FUNCTION_BLOCK ReactorLogic (* CAT Function Block Type *)
  (* Standard: 61499-2 *)
  (* Version 0.0, 6/7/2026, Schneider Electric, template *)
  PACKAGE SE.Nereda;
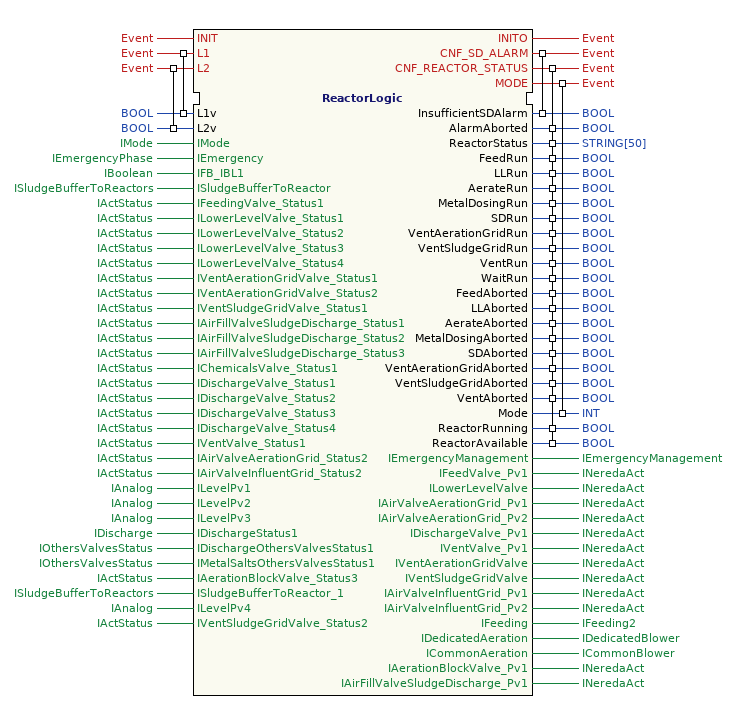
  EVENT_INPUT
    INIT;
    L1 WITH L1v;
    L2 WITH L2v;
  END_EVENT
  EVENT_OUTPUT
    INITO;
    CNF_SD_ALARM WITH InsufficientSDAlarm;
    CNF_REACTOR_STATUS WITH AlarmAborted, ReactorStatus, FeedRun, LLRun, AerateRun, MetalDosingRun, SDRun, VentAerationGridRun, VentSludgeGridRun, VentRun, WaitRun, FeedAborted, LLAborted, AerateAborted, MetalDosingAborted, SDAborted, VentAerationGridAborted, VentSludgeGridAborted, VentAborted, ReactorRunning, ReactorAvailable; (* Execution Confirmation *)
    MODE WITH Mode; (* Response from Socket *)
  END_EVENT
  VAR_INPUT
    L1v : BOOL;
    L2v : BOOL;
  END_VAR
  VAR_OUTPUT
    InsufficientSDAlarm : BOOL;
    AlarmAborted : BOOL; (* Result: IN1 OR IN2 OR ... *)
    ReactorStatus : STRING[50]; (* Output event qualifier *)
    FeedRun : BOOL;
    LLRun : BOOL;
    AerateRun : BOOL;
    MetalDosingRun : BOOL;
    SDRun : BOOL;
    VentAerationGridRun : BOOL;
    VentSludgeGridRun : BOOL;
    VentRun : BOOL;
    WaitRun : BOOL;
    FeedAborted : BOOL;
    LLAborted : BOOL;
    AerateAborted : BOOL;
    MetalDosingAborted : BOOL;
    SDAborted : BOOL;
    VentAerationGridAborted : BOOL;
    VentSludgeGridAborted : BOOL;
    VentAborted : BOOL;
    Mode : INT; (* Response Data from Socket *)
    ReactorRunning : BOOL; (* Result: IN1 OR IN2 OR ... *)
    ReactorAvailable : BOOL; (* Result: IN1 AND IN2 AND ... *)
  END_VAR
  SOCKETS
    IMode : IMode;
    IEmergency : IEmergencyPhase;
    IFB_IBL1 : IBoolean;
    ISludgeBufferToReactor : ISludgeBufferToReactors;
  END_SOCKETS
  SOCKETS
    IFeedingValve_Status1 : IActStatus; (* Phase Feed Status *)
    ILowerLevelValve_Status1 : IActStatus;
    ILowerLevelValve_Status2 : IActStatus;
    ILowerLevelValve_Status3 : IActStatus;
    ILowerLevelValve_Status4 : IActStatus;
    IVentAerationGridValve_Status1 : IActStatus;
    IVentAerationGridValve_Status2 : IActStatus; (* Phase Aerate Status *)
    IVentSludgeGridValve_Status1 : IActStatus;
    IAirFillValveSludgeDischarge_Status1 : IActStatus;
    IAirFillValveSludgeDischarge_Status2 : IActStatus;
    IAirFillValveSludgeDischarge_Status3 : IActStatus;
    IChemicalsValve_Status1 : IActStatus;
    IDischargeValve_Status1 : IActStatus; (* Phase Feed Status *)
    IDischargeValve_Status2 : IActStatus; (* Phase Sludge Discharge Status *)
    IDischargeValve_Status3 : IActStatus; (* Phase Feed Status *)
    IDischargeValve_Status4 : IActStatus; (* Phase Aerate Status *)
    IVentValve_Status1 : IActStatus; (* Phase Vent Status *)
    IAirValveAerationGrid_Status2 : IActStatus; (* Phase Vent Status *)
    IAirValveInfluentGrid_Status2 : IActStatus; (* Phase Vent Status *)
    ILevelPv1 : IAnalog; (* Phase Feed Status *)
    ILevelPv2 : IAnalog; (* Phase Aerate Status *)
    ILevelPv3 : IAnalog;
    IDischargeStatus1 : IDischarge; (* Phase Sludge Discharge Status *)
    IDischargeOthersValvesStatus1 : IOthersValvesStatus; (* Phase Sludge Discharge Status *)
    IMetalSaltsOthersValvesStatus1 : IOthersValvesStatus;
    IAerationBlockValve_Status3 : IActStatus; (* Phase Aerate Status *)
    ISludgeBufferToReactor_1 : ISludgeBufferToReactors;
    ILevelPv4 : IAnalog; (* Phase Feed Status *)
    IVentSludgeGridValve_Status2 : IActStatus;
  END_SOCKETS
  PLUGS
    IEmergencyManagement : IEmergencyManagement(pin_D997CA5474076632 := TRUE);
  END_PLUGS
  PLUGS
    IFeedValve_Pv1 : INeredaAct; (* Phase Feed Cmd *)
    ILowerLevelValve : INeredaAct;
    IAirValveAerationGrid_Pv1 : INeredaAct; (* Phase Aerate Cmd *)
    IAirValveAerationGrid_Pv2 : INeredaAct; (* Phase Vent Cmd *)
    IDischargeValve_Pv1 : INeredaAct; (* Phase Sludge Discharge Cmd *)
    IVentValve_Pv1 : INeredaAct; (* Phase Vent Cmd *)
    IVentAerationGridValve : INeredaAct;
    IVentSludgeGridValve : INeredaAct;
    IAirValveInfluentGrid_Pv1 : INeredaAct; (* Phase Aerate Cmd *)
    IAirValveInfluentGrid_Pv2 : INeredaAct; (* Phase Vent Cmd *)
    IFeeding : IFeeding2; (* Phase Feed Cmd *)
    IDedicatedAeration : IDedicatedBlower; (* Phase Aerate Cmd *)
    ICommonAeration : ICommonBlower;
    IAerationBlockValve_Pv1 : INeredaAct; (* Phase Aerate Cmd *)
    IAirFillValveSludgeDischarge_Pv1 : INeredaAct;
  END_PLUGS
  (* 01 - FUNCTIONNAL INPUT INTERFACE *)
  (* 00 - INITIALIZATION *)
  (* 05 - LOGIC *)
  (* 06 - HMI INTERFACE *)
  (* 03 - FIELD INTERFACE *)
  (* Phase Feed *)
  (* Phase Aerate *)
  (* Phase Wait *)
  (* Phase Sludge Discharge *)
  (* Phase vent *)
  (* Phase Feed *)
  (* Phase Aerate *)
  (* Phase Sludge Discharge *)
  (* Phase Vent *)
  (* Check Phase Running / Check Phase Aborted *)
  (* 02 - FUNCTIONNAL OUTPUT INTERFACE *)
  (* Phase Feed - AV4x101 *)
  (* Phase Aerate *)
  (* Phase Sludge Discharge *)
  (* Phase Vent *)
  (* Phase lower level *)
  (* Phase metal dosing *)
  (* Phase vent aeration grid *)
  (* Phase vent sludge grid *)
  (* Phase Lower Level - AV4x102 *)
  (* Phase metal dosing *)
  (* Phase Vent Aeration Grid *)
  (* Phase Vent Sludge Grid *)
  (* Phase Lower Level *)
  (* Phase Metal Dosing *)
  (* Phase VentAeration Grid *)
  (* Phase VentAeration  SLUDGE Grid *)
  (* Sufficient Feed Flow *)
  (* Actuators Tags : - Feed valve :                                  AV4x101 - Lower level valve :                        AV4x102 - Air fill valve sludge discharge :    AV4x171 - Chemicals valve :                         AV4x108 - Discharge valve :                         AV4x103 - Vent aeration grid valve :             AV4x107 - Vent sludge grid valve :               AV4x172 *)
  FBS
    Feed : Phase;
    OCFeed : FeedOC;
    Aerate : Phase;
    Wait : Phase;
    SludgeDischarge : Phase;
    Vent : Phase;
    IThis : ReactorLogic_HMI(QI := TRUE);
    LogicFeed : CmdFeed;
    OCAerate : AerateOC;
    OCVent : VentOC;
    OCSludgeDischarge : SludgeDischargeOC;
    LogicAerate : CmdAerate;
    LogicSludgeDischarge : CmdSludgeDischarge;
    LogicVent : CmdVent;
    CheckPhaseRunning : OR_201A0B5C94C9C72F7; {SET_ATTRIBUTE(Configuration.GenericFBType.InterfaceParams, Runtime.Standard#CNT:=9;OUT:BOOL)}
    CheckPhaseAborted : OR_201A0B5C94C9C72F7; {SET_ATTRIBUTE(Configuration.GenericFBType.InterfaceParams, Runtime.Standard#CNT:=9;OUT:BOOL)}
    ReactorStatusMng : ReactorStatus;
    OCWait : NoOC;
    LogicWait : NoCmd;
    NoFeedAerateAborted : NOT_425622A9A4AC6C60; {SET_ATTRIBUTE(Configuration.GenericFBType.InterfaceParams, Runtime.Standard#CNT:=2;OUT${CNT$}:BOOL,BOOL)}
    ReactorAvalable : AND_150A6959DE81880FD; {SET_ATTRIBUTE(Configuration.GenericFBType.InterfaceParams, Runtime.Standard#CNT:=5;OUT:BOOL)}
    CheckPhaseInterlocked : OR_201A0B5C94C9C72F7; {SET_ATTRIBUTE(Configuration.GenericFBType.InterfaceParams, Runtime.Standard#CNT:=9;OUT:BOOL)}
    NoForceUnavailable : NOT_42C76073DCEB1A7A; {SET_ATTRIBUTE(Configuration.GenericFBType.InterfaceParams, Runtime.Standard#CNT:=1;OUT${CNT$}:BOOL)}
    FeedAv : CmdAndIlcked;
    AerateAv : CmdAndIlcked;
    LowerLevel : Phase;
    OCLowerLevel : LowerLevelOC;
    LogicLowerLevel : CmdOneAct;
    MetalDosing : Phase;
    OCMetalDosing : MetalDosingOC;
    VentAerationGrid : Phase;
    VentSludgeGrid : Phase;
    LogicMetalDosing : NoCmd;
    LogicVentAerationGrid : CmdOneAct;
    LogicVentSludgeGrid : CmdOneAct;
    OCVentAerationGrid : VentAerationGridOC;
    SufficientFeedFlow : SufficientFeedFlow;
    OCVentSludgeGrid : VentSludgeGridOC;
  END_FBS
  EVENT_CONNECTIONS
    INIT TO IThis.7A91C2AD0F4AB044;
    IThis.DCC20F2F18497858 TO OCFeed.EEE7655ECB3D19E4;
    OCFeed.C3BD2951F6A0C2EA TO LogicFeed.413C016DFFB59D18;
    LogicFeed.B72A275F8DEDE920 TO OCLowerLevel.EEE7655ECB3D19E4;
    OCAerate.C3BD2951F6A0C2EA TO LogicAerate.413C016DFFB59D18;
    LogicMetalDosing.B72A275F8DEDE920 TO OCSludgeDischarge.EEE7655ECB3D19E4;
    OCSludgeDischarge.C3BD2951F6A0C2EA TO LogicSludgeDischarge.413C016DFFB59D18;
    OCVent.C3BD2951F6A0C2EA TO LogicVent.413C016DFFB59D18;
    LogicVent.B72A275F8DEDE920 TO OCWait.EEE7655ECB3D19E4;
    OCWait.C3BD2951F6A0C2EA TO LogicWait.413C016DFFB59D18;
    LogicWait.B72A275F8DEDE920 TO INITO;
    IMode.MODE TO LogicFeed.42062FCE2A6CF2D8;
    IEmergency.0FA2667D36826F2B TO LogicFeed.B960D5854AD6242C;
    IEmergency.BC34E8F0E0F52444 TO LogicFeed.B960D5854AD6242C;
    LogicFeed.C2051489E8C54C8C TO IEmergencyManagement.FEED_TIME;
    IMode.MODE TO Feed.8CB9CCC96FA037F2;
    IMode.RESET TO Feed.0B9CBD1FB67738FF;
    IMode.MODE TO Aerate.8CB9CCC96FA037F2;
    IMode.MODE TO SludgeDischarge.8CB9CCC96FA037F2;
    IMode.MODE TO Vent.8CB9CCC96FA037F2;
    IMode.MODE TO Wait.8CB9CCC96FA037F2;
    IMode.RESET TO Wait.0B9CBD1FB67738FF;
    IMode.RESET TO Vent.0B9CBD1FB67738FF;
    IMode.RESET TO SludgeDischarge.0B9CBD1FB67738FF;
    IMode.RESET TO Aerate.0B9CBD1FB67738FF;
    IEmergency.42529785B6820948 TO Feed.CC2F040586B1B15C;
    IEmergency.B633B7A44F850807 TO Aerate.CC2F040586B1B15C;
    IEmergency.B3BCF5E9C62C69B8 TO SludgeDischarge.CC2F040586B1B15C;
    IEmergency.ACC2803E6ACB558D TO Vent.CC2F040586B1B15C;
    IEmergency.8A3A142CC73C9F25 TO Wait.CC2F040586B1B15C;
    IEmergency.0FA2667D36826F2B TO Feed.4B853D9399632249;
    IEmergency.0FA2667D36826F2B TO Aerate.4B853D9399632249;
    IEmergency.0FA2667D36826F2B TO SludgeDischarge.4B853D9399632249;
    IEmergency.0FA2667D36826F2B TO Vent.4B853D9399632249;
    IEmergency.0FA2667D36826F2B TO Wait.4B853D9399632249;
    IMode.MODE TO LogicAerate.42062FCE2A6CF2D8;
    IMode.MODE TO LogicSludgeDischarge.42062FCE2A6CF2D8;
    IMode.MODE TO LogicVent.42062FCE2A6CF2D8;
    IEmergency.FF8E2C9D67AADBF4 TO LogicVent.4520C80B23F9200E;
    IEmergency.0FA2667D36826F2B TO LogicAerate.B960D5854AD6242C;
    IEmergency.1BDE0720AC8B4391 TO LogicAerate.B960D5854AD6242C;
    Feed.C9D225E9FF976CF5 TO IEmergency.3CBA18632C5993F7;
    Aerate.C9D225E9FF976CF5 TO IEmergency.B9A3DD1A626C862D;
    SludgeDischarge.C9D225E9FF976CF5 TO IEmergency.4DCB92F6993C5EE1;
    Vent.C9D225E9FF976CF5 TO IEmergency.3F1D0A688A5176FD;
    Wait.C9D225E9FF976CF5 TO IEmergency.B334EFD88038E789;
    L1 TO IEmergency.1F4F3B9CDE5DCB1C;
    L2 TO IEmergency.0001D958FDF5E959;
    LogicSludgeDischarge.6C61EC1722686E87 TO CNF_SD_ALARM;
    ReactorStatusMng.B6E4C96ABAEB4E2A TO IEmergencyManagement.PHASE_NO_ABORTED;
    ReactorStatusMng.B6E4C96ABAEB4E2A TO CNF_REACTOR_STATUS;
    SludgeDischarge.C9D225E9FF976CF5 TO IEmergencyManagement.SD_REACTOR;
    IMode.MODE TO IEmergencyManagement.MODE;
    IEmergency.0FA2667D36826F2B TO LogicFeed.AEFB8B0C9F8E43F1;
    IEmergency.3CAF22C03BECB249 TO LogicFeed.5AF598EEF12AFAB6;
    Aerate.C9D225E9FF976CF5 TO LogicFeed.33974E3871FD794D;
    NoFeedAerateAborted.CNF TO NoForceUnavailable.REQ;
    ReactorAvalable.CNF TO ReactorStatusMng.2C4D36E78CFC061F;
    AerateAv.F9551E9B0D43115F TO ReactorAvalable.REQ;
    NoForceUnavailable.CNF TO ReactorAvalable.REQ;
    IEmergency.42529785B6820948 TO FeedAv.42EB462001E7FF11;
    IEmergency.B633B7A44F850807 TO AerateAv.42EB462001E7FF11;
    FeedAv.F9551E9B0D43115F TO ReactorAvalable.REQ;
    IMode.MODE TO MODE;
    IEmergencyManagement.33EC5B834E8FFAF3 TO IEmergencyManagement.12FB600C11F75EA2;
    OCLowerLevel.C3BD2951F6A0C2EA TO LogicLowerLevel.413C016DFFB59D18;
    OCMetalDosing.C3BD2951F6A0C2EA TO LogicMetalDosing.413C016DFFB59D18;
    LogicAerate.B72A275F8DEDE920 TO OCMetalDosing.EEE7655ECB3D19E4;
    LogicLowerLevel.B72A275F8DEDE920 TO OCAerate.EEE7655ECB3D19E4;
    IMode.MODE TO LowerLevel.8CB9CCC96FA037F2;
    IMode.MODE TO MetalDosing.8CB9CCC96FA037F2;
    IMode.MODE TO VentAerationGrid.8CB9CCC96FA037F2;
    IMode.MODE TO VentSludgeGrid.8CB9CCC96FA037F2;
    IMode.RESET TO VentSludgeGrid.0B9CBD1FB67738FF;
    IMode.RESET TO VentAerationGrid.0B9CBD1FB67738FF;
    IMode.RESET TO MetalDosing.0B9CBD1FB67738FF;
    IMode.RESET TO LowerLevel.0B9CBD1FB67738FF;
    IEmergency.2000F66036015D52 TO LowerLevel.CC2F040586B1B15C;
    IEmergency.0FA2667D36826F2B TO LowerLevel.4B853D9399632249;
    IEmergency.0FA2667D36826F2B TO MetalDosing.4B853D9399632249;
    IEmergency.0FA2667D36826F2B TO VentAerationGrid.4B853D9399632249;
    IEmergency.0FA2667D36826F2B TO VentSludgeGrid.4B853D9399632249;
    LowerLevel.C9D225E9FF976CF5 TO IEmergency.CF95EBECB4A2EBBE;
    Feed.C9D225E9FF976CF5 TO LowerLevel.58804E595E0ACE04;
    Aerate.C9D225E9FF976CF5 TO LowerLevel.58804E595E0ACE04;
    MetalDosing.C9D225E9FF976CF5 TO LowerLevel.58804E595E0ACE04;
    SludgeDischarge.C9D225E9FF976CF5 TO LowerLevel.58804E595E0ACE04;
    VentAerationGrid.C9D225E9FF976CF5 TO LowerLevel.58804E595E0ACE04;
    VentSludgeGrid.C9D225E9FF976CF5 TO LowerLevel.58804E595E0ACE04;
    Vent.C9D225E9FF976CF5 TO LowerLevel.58804E595E0ACE04;
    Wait.C9D225E9FF976CF5 TO LowerLevel.58804E595E0ACE04;
    LowerLevel.C9D225E9FF976CF5 TO Feed.58804E595E0ACE04;
    Aerate.C9D225E9FF976CF5 TO Feed.58804E595E0ACE04;
    MetalDosing.C9D225E9FF976CF5 TO Feed.58804E595E0ACE04;
    SludgeDischarge.C9D225E9FF976CF5 TO Feed.58804E595E0ACE04;
    VentAerationGrid.C9D225E9FF976CF5 TO Feed.58804E595E0ACE04;
    VentSludgeGrid.C9D225E9FF976CF5 TO Feed.58804E595E0ACE04;
    Vent.C9D225E9FF976CF5 TO Feed.58804E595E0ACE04;
    Wait.C9D225E9FF976CF5 TO Feed.58804E595E0ACE04;
    Feed.C9D225E9FF976CF5 TO Aerate.58804E595E0ACE04;
    LowerLevel.C9D225E9FF976CF5 TO Aerate.58804E595E0ACE04;
    MetalDosing.C9D225E9FF976CF5 TO Aerate.58804E595E0ACE04;
    SludgeDischarge.C9D225E9FF976CF5 TO Aerate.58804E595E0ACE04;
    VentAerationGrid.C9D225E9FF976CF5 TO Aerate.58804E595E0ACE04;
    VentSludgeGrid.C9D225E9FF976CF5 TO Aerate.58804E595E0ACE04;
    Vent.C9D225E9FF976CF5 TO Aerate.58804E595E0ACE04;
    Wait.C9D225E9FF976CF5 TO Aerate.58804E595E0ACE04;
    Feed.C9D225E9FF976CF5 TO MetalDosing.58804E595E0ACE04;
    LowerLevel.C9D225E9FF976CF5 TO MetalDosing.58804E595E0ACE04;
    Aerate.C9D225E9FF976CF5 TO MetalDosing.58804E595E0ACE04;
    SludgeDischarge.C9D225E9FF976CF5 TO MetalDosing.58804E595E0ACE04;
    VentAerationGrid.C9D225E9FF976CF5 TO MetalDosing.58804E595E0ACE04;
    VentSludgeGrid.C9D225E9FF976CF5 TO MetalDosing.58804E595E0ACE04;
    Vent.C9D225E9FF976CF5 TO MetalDosing.58804E595E0ACE04;
    Wait.C9D225E9FF976CF5 TO MetalDosing.58804E595E0ACE04;
    Feed.C9D225E9FF976CF5 TO SludgeDischarge.58804E595E0ACE04;
    LowerLevel.C9D225E9FF976CF5 TO SludgeDischarge.58804E595E0ACE04;
    Aerate.C9D225E9FF976CF5 TO SludgeDischarge.58804E595E0ACE04;
    MetalDosing.C9D225E9FF976CF5 TO SludgeDischarge.58804E595E0ACE04;
    VentAerationGrid.C9D225E9FF976CF5 TO SludgeDischarge.58804E595E0ACE04;
    VentSludgeGrid.C9D225E9FF976CF5 TO SludgeDischarge.58804E595E0ACE04;
    Vent.C9D225E9FF976CF5 TO SludgeDischarge.58804E595E0ACE04;
    Wait.C9D225E9FF976CF5 TO SludgeDischarge.58804E595E0ACE04;
    Feed.C9D225E9FF976CF5 TO VentAerationGrid.58804E595E0ACE04;
    LowerLevel.C9D225E9FF976CF5 TO VentAerationGrid.58804E595E0ACE04;
    Aerate.C9D225E9FF976CF5 TO VentAerationGrid.58804E595E0ACE04;
    MetalDosing.C9D225E9FF976CF5 TO VentAerationGrid.58804E595E0ACE04;
    SludgeDischarge.C9D225E9FF976CF5 TO VentAerationGrid.58804E595E0ACE04;
    VentSludgeGrid.C9D225E9FF976CF5 TO VentAerationGrid.58804E595E0ACE04;
    Vent.C9D225E9FF976CF5 TO VentAerationGrid.58804E595E0ACE04;
    Wait.C9D225E9FF976CF5 TO VentAerationGrid.58804E595E0ACE04;
    Feed.C9D225E9FF976CF5 TO VentSludgeGrid.58804E595E0ACE04;
    LowerLevel.C9D225E9FF976CF5 TO VentSludgeGrid.58804E595E0ACE04;
    Aerate.C9D225E9FF976CF5 TO VentSludgeGrid.58804E595E0ACE04;
    MetalDosing.C9D225E9FF976CF5 TO VentSludgeGrid.58804E595E0ACE04;
    SludgeDischarge.C9D225E9FF976CF5 TO VentSludgeGrid.58804E595E0ACE04;
    VentAerationGrid.C9D225E9FF976CF5 TO VentSludgeGrid.58804E595E0ACE04;
    Vent.C9D225E9FF976CF5 TO VentSludgeGrid.58804E595E0ACE04;
    Wait.C9D225E9FF976CF5 TO VentSludgeGrid.58804E595E0ACE04;
    Feed.C9D225E9FF976CF5 TO Vent.58804E595E0ACE04;
    LowerLevel.C9D225E9FF976CF5 TO Vent.58804E595E0ACE04;
    Aerate.C9D225E9FF976CF5 TO Vent.58804E595E0ACE04;
    MetalDosing.C9D225E9FF976CF5 TO Vent.58804E595E0ACE04;
    SludgeDischarge.C9D225E9FF976CF5 TO Vent.58804E595E0ACE04;
    VentAerationGrid.C9D225E9FF976CF5 TO Vent.58804E595E0ACE04;
    VentSludgeGrid.C9D225E9FF976CF5 TO Vent.58804E595E0ACE04;
    Wait.C9D225E9FF976CF5 TO Vent.58804E595E0ACE04;
    LowerLevel.C9D225E9FF976CF5 TO Wait.58804E595E0ACE04;
    Aerate.C9D225E9FF976CF5 TO Wait.58804E595E0ACE04;
    Feed.C9D225E9FF976CF5 TO Wait.58804E595E0ACE04;
    MetalDosing.C9D225E9FF976CF5 TO Wait.58804E595E0ACE04;
    SludgeDischarge.C9D225E9FF976CF5 TO Wait.58804E595E0ACE04;
    VentAerationGrid.C9D225E9FF976CF5 TO Wait.58804E595E0ACE04;
    VentSludgeGrid.C9D225E9FF976CF5 TO Wait.58804E595E0ACE04;
    Vent.C9D225E9FF976CF5 TO Wait.58804E595E0ACE04;
    Feed.C9D225E9FF976CF5 TO CheckPhaseRunning.REQ;
    Aerate.C9D225E9FF976CF5 TO CheckPhaseRunning.REQ;
    SludgeDischarge.C9D225E9FF976CF5 TO CheckPhaseRunning.REQ;
    Vent.C9D225E9FF976CF5 TO CheckPhaseRunning.REQ;
    Wait.C9D225E9FF976CF5 TO CheckPhaseRunning.REQ;
    IEmergency.3CAF22C03BECB249 TO CheckPhaseRunning.REQ;
    LowerLevel.C9D225E9FF976CF5 TO CheckPhaseRunning.REQ;
    MetalDosing.C9D225E9FF976CF5 TO CheckPhaseRunning.REQ;
    VentAerationGrid.C9D225E9FF976CF5 TO CheckPhaseRunning.REQ;
    VentSludgeGrid.C9D225E9FF976CF5 TO CheckPhaseRunning.REQ;
    CheckPhaseRunning.CNF TO CheckPhaseAborted.REQ;
    CheckPhaseAborted.CNF TO CheckPhaseInterlocked.REQ;
    CheckPhaseInterlocked.CNF TO NoFeedAerateAborted.REQ;
    LogicFeed.6987DA41EB22743F TO OCLowerLevel.233986BE2644F7CE;
    LogicSludgeDischarge.B72A275F8DEDE920 TO OCVentAerationGrid.EEE7655ECB3D19E4;
    OCVentAerationGrid.C3BD2951F6A0C2EA TO LogicVentAerationGrid.413C016DFFB59D18;
    LogicVentAerationGrid.B72A275F8DEDE920 TO OCVentSludgeGrid.EEE7655ECB3D19E4;
    OCVentSludgeGrid.C3BD2951F6A0C2EA TO LogicVentSludgeGrid.413C016DFFB59D18;
    LogicVentSludgeGrid.B72A275F8DEDE920 TO OCVent.EEE7655ECB3D19E4;
    IEmergency.DAE1720DE74FAACB TO VentSludgeGrid.CC2F040586B1B15C;
    IEmergency.0F544A40694CE400 TO VentAerationGrid.CC2F040586B1B15C;
    VentSludgeGrid.C9D225E9FF976CF5 TO IEmergency.2E6F627FE71D38B1;
    IFB_IBL1.6A2938685EDB5ACB TO IEmergency.2DDA8AB533D7441D;
    Feed.53078EA27DFC2153 TO SufficientFeedFlow.4077042B95A5B675;
    Feed.C9D225E9FF976CF5 TO SufficientFeedFlow.39D7C3AFE6D016A9;
  END_CONNECTIONS
  DATA_CONNECTIONS
    IMode.Mode TO LogicFeed.359E24E45FC44765;
    IEmergency.34423AC7BCF3714C TO LogicFeed.6B6DC0CDC9D4BF59;
    LogicFeed.28A1E7F15B123DAF TO IEmergencyManagement.FeedTime;
    LogicFeed.28FA2D399946C22C TO IEmergencyManagement.CD077CD9F3BB8B76;
    IMode.Mode TO Feed.60C668C3F76389FF;
    IMode.Mode TO Aerate.60C668C3F76389FF;
    IMode.Mode TO SludgeDischarge.60C668C3F76389FF;
    IMode.Mode TO Vent.60C668C3F76389FF;
    IMode.Mode TO Wait.60C668C3F76389FF;
    IMode.Reset TO Feed.3AA98D5129903FF7;
    IMode.Reset TO Aerate.3AA98D5129903FF7;
    IMode.Reset TO SludgeDischarge.3AA98D5129903FF7;
    IMode.Reset TO Vent.3AA98D5129903FF7;
    IMode.Reset TO Wait.3AA98D5129903FF7;
    IEmergency.8B7B31E6EA54014D TO Feed.195C6B3853E1CD26;
    IEmergency.09084E8C7BADBD46 TO Aerate.195C6B3853E1CD26;
    IEmergency.C947D1396F3B0873 TO SludgeDischarge.195C6B3853E1CD26;
    IEmergency.6926B570C8BA75E8 TO Vent.195C6B3853E1CD26;
    IEmergency.C584AEAB998AB515 TO Wait.195C6B3853E1CD26;
    IEmergency.5159724764416574 TO Feed.2BB71ADCF214FB08;
    IEmergency.5159724764416574 TO Aerate.2BB71ADCF214FB08;
    IEmergency.5159724764416574 TO SludgeDischarge.2BB71ADCF214FB08;
    IEmergency.5159724764416574 TO Vent.2BB71ADCF214FB08;
    IEmergency.5159724764416574 TO Wait.2BB71ADCF214FB08;
    IMode.Mode TO LogicAerate.359E24E45FC44765;
    IMode.Mode TO LogicSludgeDischarge.359E24E45FC44765;
    IMode.Mode TO LogicVent.359E24E45FC44765;
    IEmergency.51705890CC419D73 TO LogicVent.78363E9590E65C66;
    IEmergency.F44F737D6F09989F TO LogicVent.D274A1E4F34A8A6F;
    IEmergency.5159724764416574 TO LogicAerate.FC5C6DAB9F518715;
    IEmergency.8B46E1E2CAE6076D TO LogicAerate.6B6DC0CDC9D4BF59;
    IEmergency.A29A102F17AA7B5F TO LogicAerate.646825DD30F2EA5E;
    IEmergency.EC5E58B468310216 TO LogicAerate.CAA51838933CA377;
    Feed.D4263C4F5EA880F1 TO IEmergency.599667ECF678E518;
    Feed.205C2090874C407F TO IEmergency.4F5ECA9F9BF691B9;
    Aerate.D4263C4F5EA880F1 TO IEmergency.656FC0E59D395E4C;
    Aerate.205C2090874C407F TO IEmergency.3EE993A4C10CAFA0;
    SludgeDischarge.D4263C4F5EA880F1 TO IEmergency.9CFBB312DE29B9C4;
    SludgeDischarge.205C2090874C407F TO IEmergency.9D8612C8A748A8DE;
    Vent.D4263C4F5EA880F1 TO IEmergency.E996774D431E1B79;
    Vent.205C2090874C407F TO IEmergency.6B3CB5C4C50BE958;
    Wait.D4263C4F5EA880F1 TO IEmergency.A92252B4F4DF917A;
    Wait.205C2090874C407F TO IEmergency.F87C7AE958A99541;
    L1v TO IEmergency.579DEB3758BDB938;
    L2v TO IEmergency.1156E288C0C38120;
    LogicSludgeDischarge.38484D1DA7E12332 TO InsufficientSDAlarm;
    ReactorAvalable.OUT TO IEmergencyManagement.3C69BB1A066E9338;
    IMode.Mode TO IEmergencyManagement.Mode;
    SludgeDischarge.79A84BC5970E2DB6 TO IEmergencyManagement.SDReactor;
    LogicFeed.56DD7ED30B2405EE TO IEmergencyManagement.B60AD268A06073AC;
    LogicFeed.ADD01AACDDF238E3 TO IEmergencyManagement.8FB3B1E89F73B5E3;
    ReactorStatusMng.407F4164D4F8FA5A TO ReactorStatus;
    Feed.79A84BC5970E2DB6 TO FeedRun;
    Aerate.79A84BC5970E2DB6 TO AerateRun;
    SludgeDischarge.79A84BC5970E2DB6 TO SDRun;
    Vent.79A84BC5970E2DB6 TO VentRun;
    Wait.79A84BC5970E2DB6 TO WaitRun;
    Feed.9521593C56F0BC35 TO FeedAborted;
    Aerate.9521593C56F0BC35 TO AerateAborted;
    SludgeDischarge.9521593C56F0BC35 TO SDAborted;
    Vent.9521593C56F0BC35 TO VentAborted;
    IMode.Mode TO Mode;
    ReactorAvalable.OUT TO ReactorAvailable;
    IMode.Mode TO LowerLevel.60C668C3F76389FF;
    IMode.Mode TO MetalDosing.60C668C3F76389FF;
    IMode.Mode TO VentAerationGrid.60C668C3F76389FF;
    IMode.Mode TO VentSludgeGrid.60C668C3F76389FF;
    IMode.Reset TO VentSludgeGrid.3AA98D5129903FF7;
    IMode.Reset TO VentAerationGrid.3AA98D5129903FF7;
    IMode.Reset TO MetalDosing.3AA98D5129903FF7;
    IMode.Reset TO LowerLevel.3AA98D5129903FF7;
    IEmergency.5159724764416574 TO VentSludgeGrid.2BB71ADCF214FB08;
    IEmergency.5159724764416574 TO VentAerationGrid.2BB71ADCF214FB08;
    IEmergency.5159724764416574 TO MetalDosing.2BB71ADCF214FB08;
    IEmergency.5159724764416574 TO LowerLevel.2BB71ADCF214FB08;
    LowerLevel.D4263C4F5EA880F1 TO IEmergency.A1460632301E8B7F;
    LowerLevel.205C2090874C407F TO IEmergency.9FAB21A852151825;
    Aerate.79A84BC5970E2DB6 TO IEmergency.A63167A113600EB8;
    SludgeDischarge.79A84BC5970E2DB6 TO IEmergency.28136BA3C9D3697F;
    Feed.79A84BC5970E2DB6 TO IEmergency.F208B10244BCFEF2;
    IEmergency.5159724764416574 TO LogicFeed.22CCD0256B929A29;
    IEmergency.63583CB69DED3592 TO LogicFeed.76E6DC11433E66C6;
    Aerate.D4263C4F5EA880F1 TO LogicFeed.2734297AD11954E2;
    Aerate.810982233799B264 TO LogicFeed.D164033516116A09;
    Aerate.9521593C56F0BC35 TO LogicFeed.EC40A72DA608F5D6;
    Aerate.205C2090874C407F TO LogicFeed.4A131CABC362820B;
    Feed.79A84BC5970E2DB6 TO CheckPhaseRunning.IN1;
    Aerate.79A84BC5970E2DB6 TO CheckPhaseRunning.IN3;
    SludgeDischarge.79A84BC5970E2DB6 TO CheckPhaseRunning.IN5;
    Vent.79A84BC5970E2DB6 TO CheckPhaseRunning.IN8;
    Wait.79A84BC5970E2DB6 TO CheckPhaseRunning.IN9;
    CheckPhaseRunning.OUT TO IEmergencyManagement.PhaseRun;
    CheckPhaseRunning.OUT TO ReactorStatusMng.61016BEC47180831;
    CheckPhaseRunning.OUT TO ReactorRunning;
    CheckPhaseAborted.OUT TO AlarmAborted;
    CheckPhaseAborted.OUT TO IEmergencyManagement.PhaseNoAborted;
    VentSludgeGrid.79A84BC5970E2DB6 TO CheckPhaseRunning.IN7;
    VentAerationGrid.79A84BC5970E2DB6 TO CheckPhaseRunning.IN6;
    MetalDosing.79A84BC5970E2DB6 TO CheckPhaseRunning.IN4;
    LowerLevel.79A84BC5970E2DB6 TO CheckPhaseRunning.IN2;
    Feed.9521593C56F0BC35 TO CheckPhaseAborted.IN1;
    LowerLevel.9521593C56F0BC35 TO CheckPhaseAborted.IN2;
    Aerate.9521593C56F0BC35 TO CheckPhaseAborted.IN3;
    MetalDosing.9521593C56F0BC35 TO CheckPhaseAborted.IN4;
    SludgeDischarge.9521593C56F0BC35 TO CheckPhaseAborted.IN5;
    VentAerationGrid.9521593C56F0BC35 TO CheckPhaseAborted.IN6;
    VentSludgeGrid.9521593C56F0BC35 TO CheckPhaseAborted.IN7;
    Vent.9521593C56F0BC35 TO CheckPhaseAborted.IN8;
    Wait.9521593C56F0BC35 TO CheckPhaseAborted.IN9;
    Feed.205C2090874C407F TO CheckPhaseInterlocked.IN1;
    LowerLevel.205C2090874C407F TO CheckPhaseInterlocked.IN2;
    Aerate.205C2090874C407F TO CheckPhaseInterlocked.IN3;
    MetalDosing.205C2090874C407F TO CheckPhaseInterlocked.IN4;
    SludgeDischarge.205C2090874C407F TO CheckPhaseInterlocked.IN5;
    VentAerationGrid.205C2090874C407F TO CheckPhaseInterlocked.IN6;
    VentSludgeGrid.205C2090874C407F TO CheckPhaseInterlocked.IN7;
    Vent.205C2090874C407F TO CheckPhaseInterlocked.IN8;
    Wait.205C2090874C407F TO CheckPhaseInterlocked.IN9;
    Feed.9521593C56F0BC35 TO NoFeedAerateAborted.IN1;
    Aerate.9521593C56F0BC35 TO NoFeedAerateAborted.IN2;
    NoFeedAerateAborted.OUT1 TO ReactorAvalable.IN1;
    NoFeedAerateAborted.OUT2 TO ReactorAvalable.IN3;
    IEmergency.63583CB69DED3592 TO NoForceUnavailable.IN1;
    NoForceUnavailable.OUT1 TO ReactorAvalable.IN2;
    FeedAv.11AB35620A02C8A5 TO ReactorAvalable.IN4;
    AerateAv.11AB35620A02C8A5 TO ReactorAvalable.IN5;
    CheckPhaseAborted.OUT TO ReactorStatusMng.E9087AE335C18478;
    IEmergency.09084E8C7BADBD46 TO AerateAv.40D3CD6CB4F43C33;
    Aerate.205C2090874C407F TO AerateAv.FDADF7D226C9DBAE;
    IEmergency.8B7B31E6EA54014D TO FeedAv.40D3CD6CB4F43C33;
    Feed.205C2090874C407F TO FeedAv.FDADF7D226C9DBAE;
    LowerLevel.D4263C4F5EA880F1 TO Feed.16DE804EA64A73FD;
    LowerLevel.9521593C56F0BC35 TO Feed.8AE7594594AA7DBB;
    LowerLevel.205C2090874C407F TO Feed.581756FA5F2310B2;
    Aerate.D4263C4F5EA880F1 TO Feed.B37A38F8606552EE;
    Aerate.9521593C56F0BC35 TO Feed.EFE2D0D8BEEEE5A1;
    Aerate.205C2090874C407F TO Feed.130A7AF73C88FF3B;
    MetalDosing.D4263C4F5EA880F1 TO Feed.2E1C72C6FFE1DB32;
    MetalDosing.9521593C56F0BC35 TO Feed.79BC17E07AAF4958;
    MetalDosing.205C2090874C407F TO Feed.8FB896B12AF28D8B;
    SludgeDischarge.D4263C4F5EA880F1 TO Feed.1BD1F2CFEE95F6A5;
    SludgeDischarge.9521593C56F0BC35 TO Feed.1927A9E54402DC97;
    SludgeDischarge.205C2090874C407F TO Feed.86D550500F595BC7;
    VentAerationGrid.D4263C4F5EA880F1 TO Feed.1B510EDDF5D546F5;
    VentAerationGrid.9521593C56F0BC35 TO Feed.97F3F66A1A366C75;
    VentAerationGrid.205C2090874C407F TO Feed.21AF629810CE5EE7;
    VentSludgeGrid.D4263C4F5EA880F1 TO Feed.9D4B2FB69B2D5F36;
    VentSludgeGrid.9521593C56F0BC35 TO Feed.501BF1423E0C07B2;
    VentSludgeGrid.205C2090874C407F TO Feed.E867FE48FC282519;
    Vent.D4263C4F5EA880F1 TO Feed.849C64AA69D74C13;
    Vent.9521593C56F0BC35 TO Feed.187BD32FC73E485F;
    Vent.205C2090874C407F TO Feed.88B46CCE0587A02F;
    Wait.D4263C4F5EA880F1 TO Feed.651C9839994E839D;
    Wait.9521593C56F0BC35 TO Feed.96E5B6CA319D8801;
    Wait.205C2090874C407F TO Feed.DCE8166438BBBF9A;
    Feed.D4263C4F5EA880F1 TO LowerLevel.16DE804EA64A73FD;
    Feed.9521593C56F0BC35 TO LowerLevel.8AE7594594AA7DBB;
    Feed.205C2090874C407F TO LowerLevel.581756FA5F2310B2;
    Aerate.D4263C4F5EA880F1 TO LowerLevel.B37A38F8606552EE;
    Aerate.9521593C56F0BC35 TO LowerLevel.EFE2D0D8BEEEE5A1;
    Aerate.205C2090874C407F TO LowerLevel.130A7AF73C88FF3B;
    MetalDosing.D4263C4F5EA880F1 TO LowerLevel.2E1C72C6FFE1DB32;
    MetalDosing.9521593C56F0BC35 TO LowerLevel.79BC17E07AAF4958;
    MetalDosing.205C2090874C407F TO LowerLevel.8FB896B12AF28D8B;
    SludgeDischarge.D4263C4F5EA880F1 TO LowerLevel.1BD1F2CFEE95F6A5;
    SludgeDischarge.9521593C56F0BC35 TO LowerLevel.1927A9E54402DC97;
    SludgeDischarge.205C2090874C407F TO LowerLevel.86D550500F595BC7;
    VentAerationGrid.D4263C4F5EA880F1 TO LowerLevel.1B510EDDF5D546F5;
    VentAerationGrid.9521593C56F0BC35 TO LowerLevel.97F3F66A1A366C75;
    VentAerationGrid.205C2090874C407F TO LowerLevel.21AF629810CE5EE7;
    VentSludgeGrid.D4263C4F5EA880F1 TO LowerLevel.9D4B2FB69B2D5F36;
    VentSludgeGrid.9521593C56F0BC35 TO LowerLevel.501BF1423E0C07B2;
    VentSludgeGrid.205C2090874C407F TO LowerLevel.E867FE48FC282519;
    Vent.D4263C4F5EA880F1 TO LowerLevel.849C64AA69D74C13;
    Vent.9521593C56F0BC35 TO LowerLevel.187BD32FC73E485F;
    Vent.205C2090874C407F TO LowerLevel.88B46CCE0587A02F;
    Wait.D4263C4F5EA880F1 TO LowerLevel.651C9839994E839D;
    Wait.9521593C56F0BC35 TO LowerLevel.96E5B6CA319D8801;
    Wait.205C2090874C407F TO LowerLevel.DCE8166438BBBF9A;
    Feed.D4263C4F5EA880F1 TO Aerate.16DE804EA64A73FD;
    Feed.9521593C56F0BC35 TO Aerate.8AE7594594AA7DBB;
    Feed.205C2090874C407F TO Aerate.581756FA5F2310B2;
    LowerLevel.D4263C4F5EA880F1 TO Aerate.B37A38F8606552EE;
    LowerLevel.9521593C56F0BC35 TO Aerate.EFE2D0D8BEEEE5A1;
    LowerLevel.205C2090874C407F TO Aerate.130A7AF73C88FF3B;
    MetalDosing.D4263C4F5EA880F1 TO Aerate.2E1C72C6FFE1DB32;
    MetalDosing.9521593C56F0BC35 TO Aerate.79BC17E07AAF4958;
    MetalDosing.205C2090874C407F TO Aerate.8FB896B12AF28D8B;
    SludgeDischarge.D4263C4F5EA880F1 TO Aerate.1BD1F2CFEE95F6A5;
    SludgeDischarge.9521593C56F0BC35 TO Aerate.1927A9E54402DC97;
    SludgeDischarge.205C2090874C407F TO Aerate.86D550500F595BC7;
    VentAerationGrid.D4263C4F5EA880F1 TO Aerate.1B510EDDF5D546F5;
    VentAerationGrid.9521593C56F0BC35 TO Aerate.97F3F66A1A366C75;
    VentAerationGrid.205C2090874C407F TO Aerate.21AF629810CE5EE7;
    VentSludgeGrid.D4263C4F5EA880F1 TO Aerate.9D4B2FB69B2D5F36;
    VentSludgeGrid.9521593C56F0BC35 TO Aerate.501BF1423E0C07B2;
    VentSludgeGrid.205C2090874C407F TO Aerate.E867FE48FC282519;
    Vent.D4263C4F5EA880F1 TO Aerate.849C64AA69D74C13;
    Vent.9521593C56F0BC35 TO Aerate.187BD32FC73E485F;
    Vent.205C2090874C407F TO Aerate.88B46CCE0587A02F;
    Wait.D4263C4F5EA880F1 TO Aerate.651C9839994E839D;
    Wait.9521593C56F0BC35 TO Aerate.96E5B6CA319D8801;
    Wait.205C2090874C407F TO Aerate.DCE8166438BBBF9A;
    Feed.D4263C4F5EA880F1 TO MetalDosing.16DE804EA64A73FD;
    Feed.9521593C56F0BC35 TO MetalDosing.8AE7594594AA7DBB;
    Feed.205C2090874C407F TO MetalDosing.581756FA5F2310B2;
    LowerLevel.D4263C4F5EA880F1 TO MetalDosing.B37A38F8606552EE;
    LowerLevel.9521593C56F0BC35 TO MetalDosing.EFE2D0D8BEEEE5A1;
    LowerLevel.205C2090874C407F TO MetalDosing.130A7AF73C88FF3B;
    Aerate.D4263C4F5EA880F1 TO MetalDosing.2E1C72C6FFE1DB32;
    Aerate.9521593C56F0BC35 TO MetalDosing.79BC17E07AAF4958;
    Aerate.205C2090874C407F TO MetalDosing.8FB896B12AF28D8B;
    SludgeDischarge.D4263C4F5EA880F1 TO MetalDosing.1BD1F2CFEE95F6A5;
    SludgeDischarge.9521593C56F0BC35 TO MetalDosing.1927A9E54402DC97;
    SludgeDischarge.205C2090874C407F TO MetalDosing.86D550500F595BC7;
    VentAerationGrid.D4263C4F5EA880F1 TO MetalDosing.1B510EDDF5D546F5;
    VentAerationGrid.9521593C56F0BC35 TO MetalDosing.97F3F66A1A366C75;
    VentAerationGrid.205C2090874C407F TO MetalDosing.21AF629810CE5EE7;
    VentSludgeGrid.D4263C4F5EA880F1 TO MetalDosing.9D4B2FB69B2D5F36;
    VentSludgeGrid.9521593C56F0BC35 TO MetalDosing.501BF1423E0C07B2;
    VentSludgeGrid.205C2090874C407F TO MetalDosing.E867FE48FC282519;
    Vent.D4263C4F5EA880F1 TO MetalDosing.849C64AA69D74C13;
    Vent.9521593C56F0BC35 TO MetalDosing.187BD32FC73E485F;
    Vent.205C2090874C407F TO MetalDosing.88B46CCE0587A02F;
    Wait.D4263C4F5EA880F1 TO MetalDosing.651C9839994E839D;
    Wait.9521593C56F0BC35 TO MetalDosing.96E5B6CA319D8801;
    Wait.205C2090874C407F TO MetalDosing.DCE8166438BBBF9A;
    Feed.D4263C4F5EA880F1 TO SludgeDischarge.16DE804EA64A73FD;
    Feed.9521593C56F0BC35 TO SludgeDischarge.8AE7594594AA7DBB;
    Feed.205C2090874C407F TO SludgeDischarge.581756FA5F2310B2;
    LowerLevel.D4263C4F5EA880F1 TO SludgeDischarge.B37A38F8606552EE;
    LowerLevel.9521593C56F0BC35 TO SludgeDischarge.EFE2D0D8BEEEE5A1;
    LowerLevel.205C2090874C407F TO SludgeDischarge.130A7AF73C88FF3B;
    Aerate.D4263C4F5EA880F1 TO SludgeDischarge.2E1C72C6FFE1DB32;
    Aerate.9521593C56F0BC35 TO SludgeDischarge.79BC17E07AAF4958;
    Aerate.205C2090874C407F TO SludgeDischarge.8FB896B12AF28D8B;
    MetalDosing.D4263C4F5EA880F1 TO SludgeDischarge.1BD1F2CFEE95F6A5;
    MetalDosing.9521593C56F0BC35 TO SludgeDischarge.1927A9E54402DC97;
    MetalDosing.205C2090874C407F TO SludgeDischarge.86D550500F595BC7;
    VentAerationGrid.D4263C4F5EA880F1 TO SludgeDischarge.1B510EDDF5D546F5;
    VentAerationGrid.9521593C56F0BC35 TO SludgeDischarge.97F3F66A1A366C75;
    VentAerationGrid.205C2090874C407F TO SludgeDischarge.21AF629810CE5EE7;
    VentSludgeGrid.D4263C4F5EA880F1 TO SludgeDischarge.9D4B2FB69B2D5F36;
    VentSludgeGrid.9521593C56F0BC35 TO SludgeDischarge.501BF1423E0C07B2;
    VentSludgeGrid.205C2090874C407F TO SludgeDischarge.E867FE48FC282519;
    Vent.D4263C4F5EA880F1 TO SludgeDischarge.849C64AA69D74C13;
    Vent.9521593C56F0BC35 TO SludgeDischarge.187BD32FC73E485F;
    Vent.205C2090874C407F TO SludgeDischarge.88B46CCE0587A02F;
    Wait.D4263C4F5EA880F1 TO SludgeDischarge.651C9839994E839D;
    Wait.9521593C56F0BC35 TO SludgeDischarge.96E5B6CA319D8801;
    Wait.205C2090874C407F TO SludgeDischarge.DCE8166438BBBF9A;
    Feed.D4263C4F5EA880F1 TO VentAerationGrid.16DE804EA64A73FD;
    Feed.9521593C56F0BC35 TO VentAerationGrid.8AE7594594AA7DBB;
    Feed.205C2090874C407F TO VentAerationGrid.581756FA5F2310B2;
    LowerLevel.D4263C4F5EA880F1 TO VentAerationGrid.B37A38F8606552EE;
    LowerLevel.9521593C56F0BC35 TO VentAerationGrid.EFE2D0D8BEEEE5A1;
    LowerLevel.205C2090874C407F TO VentAerationGrid.130A7AF73C88FF3B;
    Aerate.D4263C4F5EA880F1 TO VentAerationGrid.2E1C72C6FFE1DB32;
    Aerate.9521593C56F0BC35 TO VentAerationGrid.79BC17E07AAF4958;
    Aerate.205C2090874C407F TO VentAerationGrid.8FB896B12AF28D8B;
    MetalDosing.D4263C4F5EA880F1 TO VentAerationGrid.1BD1F2CFEE95F6A5;
    MetalDosing.9521593C56F0BC35 TO VentAerationGrid.1927A9E54402DC97;
    MetalDosing.205C2090874C407F TO VentAerationGrid.86D550500F595BC7;
    SludgeDischarge.D4263C4F5EA880F1 TO VentAerationGrid.1B510EDDF5D546F5;
    SludgeDischarge.9521593C56F0BC35 TO VentAerationGrid.97F3F66A1A366C75;
    SludgeDischarge.205C2090874C407F TO VentAerationGrid.21AF629810CE5EE7;
    VentSludgeGrid.D4263C4F5EA880F1 TO VentAerationGrid.9D4B2FB69B2D5F36;
    VentSludgeGrid.9521593C56F0BC35 TO VentAerationGrid.501BF1423E0C07B2;
    VentSludgeGrid.205C2090874C407F TO VentAerationGrid.E867FE48FC282519;
    Vent.D4263C4F5EA880F1 TO VentAerationGrid.849C64AA69D74C13;
    Vent.9521593C56F0BC35 TO VentAerationGrid.187BD32FC73E485F;
    Vent.205C2090874C407F TO VentAerationGrid.88B46CCE0587A02F;
    Wait.D4263C4F5EA880F1 TO VentAerationGrid.651C9839994E839D;
    Wait.9521593C56F0BC35 TO VentAerationGrid.96E5B6CA319D8801;
    Wait.205C2090874C407F TO VentAerationGrid.DCE8166438BBBF9A;
    Feed.D4263C4F5EA880F1 TO VentSludgeGrid.16DE804EA64A73FD;
    Feed.9521593C56F0BC35 TO VentSludgeGrid.8AE7594594AA7DBB;
    Feed.205C2090874C407F TO VentSludgeGrid.581756FA5F2310B2;
    LowerLevel.D4263C4F5EA880F1 TO VentSludgeGrid.B37A38F8606552EE;
    LowerLevel.9521593C56F0BC35 TO VentSludgeGrid.EFE2D0D8BEEEE5A1;
    LowerLevel.205C2090874C407F TO VentSludgeGrid.130A7AF73C88FF3B;
    Aerate.D4263C4F5EA880F1 TO VentSludgeGrid.2E1C72C6FFE1DB32;
    Aerate.9521593C56F0BC35 TO VentSludgeGrid.79BC17E07AAF4958;
    Aerate.205C2090874C407F TO VentSludgeGrid.8FB896B12AF28D8B;
    MetalDosing.D4263C4F5EA880F1 TO VentSludgeGrid.1BD1F2CFEE95F6A5;
    MetalDosing.9521593C56F0BC35 TO VentSludgeGrid.1927A9E54402DC97;
    MetalDosing.205C2090874C407F TO VentSludgeGrid.86D550500F595BC7;
    SludgeDischarge.D4263C4F5EA880F1 TO VentSludgeGrid.1B510EDDF5D546F5;
    SludgeDischarge.9521593C56F0BC35 TO VentSludgeGrid.97F3F66A1A366C75;
    SludgeDischarge.205C2090874C407F TO VentSludgeGrid.21AF629810CE5EE7;
    VentAerationGrid.D4263C4F5EA880F1 TO VentSludgeGrid.9D4B2FB69B2D5F36;
    VentAerationGrid.9521593C56F0BC35 TO VentSludgeGrid.501BF1423E0C07B2;
    VentAerationGrid.205C2090874C407F TO VentSludgeGrid.E867FE48FC282519;
    Vent.D4263C4F5EA880F1 TO VentSludgeGrid.849C64AA69D74C13;
    Vent.9521593C56F0BC35 TO VentSludgeGrid.187BD32FC73E485F;
    Vent.205C2090874C407F TO VentSludgeGrid.88B46CCE0587A02F;
    Wait.D4263C4F5EA880F1 TO VentSludgeGrid.651C9839994E839D;
    Wait.9521593C56F0BC35 TO VentSludgeGrid.96E5B6CA319D8801;
    Wait.205C2090874C407F TO VentSludgeGrid.DCE8166438BBBF9A;
    Feed.D4263C4F5EA880F1 TO Vent.16DE804EA64A73FD;
    Feed.9521593C56F0BC35 TO Vent.8AE7594594AA7DBB;
    Feed.205C2090874C407F TO Vent.581756FA5F2310B2;
    LowerLevel.D4263C4F5EA880F1 TO Vent.B37A38F8606552EE;
    LowerLevel.9521593C56F0BC35 TO Vent.EFE2D0D8BEEEE5A1;
    LowerLevel.205C2090874C407F TO Vent.130A7AF73C88FF3B;
    Aerate.D4263C4F5EA880F1 TO Vent.2E1C72C6FFE1DB32;
    Aerate.9521593C56F0BC35 TO Vent.79BC17E07AAF4958;
    Aerate.205C2090874C407F TO Vent.8FB896B12AF28D8B;
    MetalDosing.D4263C4F5EA880F1 TO Vent.1BD1F2CFEE95F6A5;
    MetalDosing.9521593C56F0BC35 TO Vent.1927A9E54402DC97;
    MetalDosing.205C2090874C407F TO Vent.86D550500F595BC7;
    SludgeDischarge.D4263C4F5EA880F1 TO Vent.1B510EDDF5D546F5;
    SludgeDischarge.9521593C56F0BC35 TO Vent.97F3F66A1A366C75;
    SludgeDischarge.205C2090874C407F TO Vent.21AF629810CE5EE7;
    VentAerationGrid.D4263C4F5EA880F1 TO Vent.9D4B2FB69B2D5F36;
    VentAerationGrid.9521593C56F0BC35 TO Vent.501BF1423E0C07B2;
    VentAerationGrid.205C2090874C407F TO Vent.E867FE48FC282519;
    VentSludgeGrid.D4263C4F5EA880F1 TO Vent.849C64AA69D74C13;
    VentSludgeGrid.9521593C56F0BC35 TO Vent.187BD32FC73E485F;
    VentSludgeGrid.205C2090874C407F TO Vent.88B46CCE0587A02F;
    Wait.D4263C4F5EA880F1 TO Vent.651C9839994E839D;
    Wait.9521593C56F0BC35 TO Vent.96E5B6CA319D8801;
    Wait.205C2090874C407F TO Vent.DCE8166438BBBF9A;
    Feed.D4263C4F5EA880F1 TO Wait.16DE804EA64A73FD;
    Feed.9521593C56F0BC35 TO Wait.8AE7594594AA7DBB;
    Feed.205C2090874C407F TO Wait.581756FA5F2310B2;
    LowerLevel.D4263C4F5EA880F1 TO Wait.B37A38F8606552EE;
    LowerLevel.9521593C56F0BC35 TO Wait.EFE2D0D8BEEEE5A1;
    LowerLevel.205C2090874C407F TO Wait.130A7AF73C88FF3B;
    Aerate.D4263C4F5EA880F1 TO Wait.2E1C72C6FFE1DB32;
    Aerate.9521593C56F0BC35 TO Wait.79BC17E07AAF4958;
    Aerate.205C2090874C407F TO Wait.8FB896B12AF28D8B;
    MetalDosing.D4263C4F5EA880F1 TO Wait.1BD1F2CFEE95F6A5;
    MetalDosing.9521593C56F0BC35 TO Wait.1927A9E54402DC97;
    MetalDosing.205C2090874C407F TO Wait.86D550500F595BC7;
    SludgeDischarge.D4263C4F5EA880F1 TO Wait.1B510EDDF5D546F5;
    SludgeDischarge.9521593C56F0BC35 TO Wait.97F3F66A1A366C75;
    SludgeDischarge.205C2090874C407F TO Wait.21AF629810CE5EE7;
    VentAerationGrid.D4263C4F5EA880F1 TO Wait.9D4B2FB69B2D5F36;
    VentAerationGrid.9521593C56F0BC35 TO Wait.501BF1423E0C07B2;
    VentAerationGrid.205C2090874C407F TO Wait.E867FE48FC282519;
    VentSludgeGrid.D4263C4F5EA880F1 TO Wait.849C64AA69D74C13;
    VentSludgeGrid.9521593C56F0BC35 TO Wait.187BD32FC73E485F;
    VentSludgeGrid.205C2090874C407F TO Wait.88B46CCE0587A02F;
    Vent.D4263C4F5EA880F1 TO Wait.651C9839994E839D;
    Vent.9521593C56F0BC35 TO Wait.96E5B6CA319D8801;
    Vent.205C2090874C407F TO Wait.DCE8166438BBBF9A;
    LogicFeed.1132E9FF8BB2E313 TO OCLowerLevel.4D4FA1E64F4224A7;
    LogicFeed.386D4C970C9A58D0 TO OCLowerLevel.C9CDCA69CB019B01;
    LowerLevel.79A84BC5970E2DB6 TO LLRun;
    MetalDosing.79A84BC5970E2DB6 TO MetalDosingRun;
    VentAerationGrid.79A84BC5970E2DB6 TO VentAerationGridRun;
    VentSludgeGrid.79A84BC5970E2DB6 TO VentSludgeGridRun;
    LowerLevel.9521593C56F0BC35 TO LLAborted;
    MetalDosing.9521593C56F0BC35 TO MetalDosingAborted;
    VentAerationGrid.9521593C56F0BC35 TO VentAerationGridAborted;
    VentSludgeGrid.9521593C56F0BC35 TO VentSludgeGridAborted;
    IEmergency.419E697BA1D2FB08 TO LowerLevel.195C6B3853E1CD26;
    IEmergency.486306180C62B9EF TO VentSludgeGrid.195C6B3853E1CD26;
    IEmergency.198FB8D9804ED082 TO VentAerationGrid.195C6B3853E1CD26;
    VentSludgeGrid.205C2090874C407F TO IEmergency.6531F3B6F766BAF5;
    VentSludgeGrid.D4263C4F5EA880F1 TO IEmergency.800D089965342DF6;
    LowerLevel.810982233799B264 TO IEmergency.D62F1904A2304A82;
    LowerLevel.0EEF2A6CD1053E7B TO IEmergency.EDD981DC30DF57BC;
    LowerLevel.9521593C56F0BC35 TO IEmergency.DA119668EC2B3E62;
    IFB_IBL1.12C123CBE763A47D TO IEmergency.C54C3886CAD71D0C;
    Feed.8EC98330761B0803 TO SufficientFeedFlow.00FEDE980413A29F;
    Feed.79A84BC5970E2DB6 TO SufficientFeedFlow.ADA40559F28F1824;
  END_CONNECTIONS
  ADAPTER_CONNECTIONS
    ILevelPv1 TO OCFeed.8FA4D2ED1552419F;
    IDischargeValve_Status1 TO OCFeed.C9DB6B9CC2C2B4BD;
    IFeedingValve_Status1 TO OCFeed.B074EF3F5F1CEEF8;
    ILevelPv2 TO OCAerate.8FA4D2ED1552419F;
    IVentAerationGridValve_Status2 TO OCAerate.C9DB6B9CC2C2B4BD;
    IDischargeValve_Status4 TO OCAerate.B074EF3F5F1CEEF8;
    IDischargeValve_Status2 TO OCSludgeDischarge.C9DB6B9CC2C2B4BD;
    IDischargeStatus1 TO OCSludgeDischarge.571AE691759419DA;
    IDischargeOthersValvesStatus1 TO OCSludgeDischarge.9732A0243A4ACE4A;
    ILevelPv3 TO LogicSludgeDischarge.C71A17A8E191C946;
    IAirValveAerationGrid_Status2 TO OCVent.C9DB6B9CC2C2B4BD;
    IVentValve_Status1 TO OCVent.3304055A40A11E39;
    IAirValveInfluentGrid_Status2 TO OCVent.9173AB2E31CC139F;
    OCVent.6B4386AEC7382B88 TO Vent.D86321A6D374FA01;
    Vent.84E547B453517565 TO LogicVent.E1021AA83C1C4121;
    LogicFeed.49A5E6149F21D49E TO IFeedValve_Pv1;
    LogicFeed.4D90656E0B6D5674 TO IFeeding;
    LogicAerate.09761DB05C329D8C TO IDedicatedAeration;
    LogicAerate.8BAD2B461FDE47FD TO ICommonAeration;
    LogicAerate.2A7255337C32A65B TO IAirValveAerationGrid_Pv1;
    LogicAerate.53EE01F26AD9A410 TO IAirValveInfluentGrid_Pv1;
    LogicSludgeDischarge.93DA7223BE633380 TO IDischargeValve_Pv1;
    LogicVent.2A7255337C32A65B TO IAirValveAerationGrid_Pv2;
    LogicVent.53EE01F26AD9A410 TO IVentValve_Pv1;
    LogicVent.379967A0469466F4 TO IAirValveInfluentGrid_Pv2;
    OCFeed.6B4386AEC7382B88 TO Feed.D86321A6D374FA01;
    Feed.84E547B453517565 TO LogicFeed.E1021AA83C1C4121;
    OCLowerLevel.6B4386AEC7382B88 TO LowerLevel.D86321A6D374FA01;
    LowerLevel.84E547B453517565 TO LogicLowerLevel.E1021AA83C1C4121;
    OCAerate.6B4386AEC7382B88 TO Aerate.D86321A6D374FA01;
    Aerate.84E547B453517565 TO LogicAerate.E1021AA83C1C4121;
    OCMetalDosing.6B4386AEC7382B88 TO MetalDosing.D86321A6D374FA01;
    OCSludgeDischarge.6B4386AEC7382B88 TO SludgeDischarge.D86321A6D374FA01;
    SludgeDischarge.84E547B453517565 TO LogicSludgeDischarge.E1021AA83C1C4121;
    Wait.84E547B453517565 TO LogicWait.E1021AA83C1C4121;
    OCWait.6B4386AEC7382B88 TO Wait.D86321A6D374FA01;
    MetalDosing.84E547B453517565 TO LogicMetalDosing.E1021AA83C1C4121;
    Aerate.0B38F2DD5BDB097B TO OCAerate.D1301D4825F0A59F;
    LogicLowerLevel.93DA7223BE633380 TO ILowerLevelValve;
    ILowerLevelValve_Status1 TO OCLowerLevel.C9DB6B9CC2C2B4BD;
    IDischargeValve_Status3 TO OCLowerLevel.3304055A40A11E39;
    VentAerationGrid.84E547B453517565 TO LogicVentAerationGrid.E1021AA83C1C4121;
    LogicVentAerationGrid.93DA7223BE633380 TO IVentAerationGridValve;
    VentSludgeGrid.84E547B453517565 TO LogicVentSludgeGrid.E1021AA83C1C4121;
    LogicVentSludgeGrid.93DA7223BE633380 TO IVentSludgeGridValve;
    OCVentAerationGrid.6B4386AEC7382B88 TO VentAerationGrid.D86321A6D374FA01;
    OCVentSludgeGrid.6B4386AEC7382B88 TO VentSludgeGrid.D86321A6D374FA01;
    ILowerLevelValve_Status2 TO OCFeed.EE5B0B65D6263231;
    IAirFillValveSludgeDischarge_Status1 TO OCAerate.01B8940CD7F6BC00;
    IVentSludgeGridValve_Status1 TO OCAerate.A39119FECB59F5BB;
    ILowerLevelValve_Status3 TO OCAerate.11AC25E1BE703EB6;
    IChemicalsValve_Status1 TO OCMetalDosing.C9DB6B9CC2C2B4BD;
    IMetalSaltsOthersValvesStatus1 TO OCMetalDosing.CC5D6C1B806C866F;
    ILowerLevelValve_Status4 TO OCSludgeDischarge.798232D3C4963786;
    IAirFillValveSludgeDischarge_Status2 TO OCSludgeDischarge.6AE66C2F6F3BE267;
    IVentAerationGridValve_Status1 TO OCVentAerationGrid.C9DB6B9CC2C2B4BD;
    IAerationBlockValve_Status3 TO OCAerate.9FE5D245E3D130B5;
    LogicAerate.B83F7840435E836E TO IAerationBlockValve_Pv1;
    LogicAerate.D2FE623904FAC0C3 TO IAirFillValveSludgeDischarge_Pv1;
    ISludgeBufferToReactor_1 TO OCSludgeDischarge.E347963A87AADE73;
    ILevelPv4 TO SufficientFeedFlow.C6809F86205722F6;
    SufficientFeedFlow.E7EF8DDBE5FFFE77 TO OCFeed.0E6BE92FA440258D;
    IAirFillValveSludgeDischarge_Status3 TO OCVentSludgeGrid.3304055A40A11E39;
    IVentSludgeGridValve_Status2 TO OCVentSludgeGrid.C9DB6B9CC2C2B4BD;
  END_CONNECTIONS
END_FUNCTION_BLOCK
